// TIA Portal project "SkarabeuszURC" (V11)

(* hardware
DEVICE "SIMATIC 1200 station_1"  S71200.Device
   slot 0: "S7-1200 rack"  Rack  V1.0
   slot 1: "PLC_1"  CPU 1215C DC/DC/DC  6ES7 215-1AG31-0XB0  V3.0
   slot 2: "AI4 x 13 bits / AQ2 x 14 bits_1"  6ES7 234-4HE30-0XB0  V1.0
*)

// ===== PLC "PLC_1"  CPU 1215C DC/DC/DC =====

VAR_GLOBAL   // PLC tag table "Default tag table"
   "Tag_1" AT %QW0 : Word;
END_VAR

VAR_GLOBAL   // PLC tag table "Motor_Tags"
   "Motor_1_Pin_1" AT %Q0.0 : Bool;
   "Motor_1_Pin_2" AT %Q0.1 : Bool;
   "Motor_2_Pin_1" AT %Q0.2 : Bool;
   "Motor_2_Pin_2" AT %Q0.3 : Bool;
   "Motor_1_Analog" AT %QW96 : Int;
   "Motor_2_Analog" AT %QW98 : Int;
   "Motor_T_Pin_1" AT %Q0.4 : Bool;
   "Motor_T_Pin_2" AT %Q0.5 : Bool;
END_VAR

DATA_BLOCK "ModbusData"   // DB1
{ S7_Optimized_Access := 'FALSE' }
VERSION : 0.1
   VAR
      Registers : Array [1 .. 127] of Int;
      NDR : Bool;
      DR : Bool;
      ERROR : Bool;
      DISCONNECT : Bool;
      STATUS : Word;
   END_VAR
BEGIN
END_DATA_BLOCK

DATA_BLOCK "GlobalData"   // DB3
{ S7_Optimized_Access := 'FALSE' }
VERSION : 0.1
   VAR
      Motor_1_Direction : Word;
      Motor_2_Direction : Word;
      Motor_1_Speed : Word;
      Motor_2_Speed : Word;
      Motor_Turning_Direction : Word;
      Encoder_1_Data : Word;
      Encoder_2_Data : Word;
      Edge_1_Switch : Word;
      Edge_2_Switch : Word;
   END_VAR
   VAR RETAIN
      Forward_Direction : Word := 1;
   END_VAR
   VAR
      Backward_Direction : Word := 2;
      Break_Direction : Word := 3;
      Idle_Direction : Word := 4;
      Right_Turn : Word := 5;
      Left_Turn : Word := 6;
   END_VAR
BEGIN
END_DATA_BLOCK

// folder: System blocks/Program resources

DATA_BLOCK "IEC_Timer_0_DB_1"   // DB5
{ S7_Optimized_Access := 'FALSE' }
AUTHOR : Simatic
FAMILY : IEC
NAME : IEC_TMR
VERSION : 1.0
// stored: InstanceOfName ?
"?"
BEGIN
END_DATA_BLOCK

// folder: (top level)

FUNCTION "ModbusTCP" : Void   // FC1, LAD
{ S7_Optimized_Access := 'FALSE' }
VERSION : 0.1
BEGIN

REGION Network 1
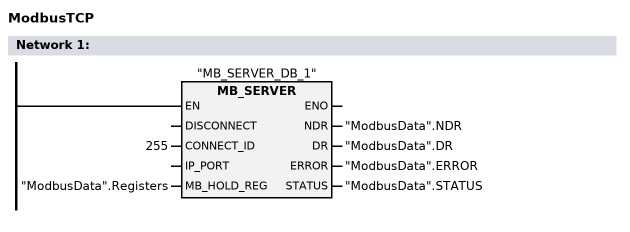
   "MB_SERVER_DB_1"(CONNECT_ID := 255,   // MB_SERVER
                    MB_HOLD_REG := "ModbusData".Registers,
                    NDR => "ModbusData".NDR,
                    DR => "ModbusData".DR,
                    ERROR => "ModbusData".ERROR,
                    STATUS => "ModbusData".STATUS);
END_REGION
END_FUNCTION

FUNCTION "Mapping" : Void   // FC2, LAD
{ S7_Optimized_Access := 'FALSE' }
VERSION : 0.1
BEGIN

REGION Network 1
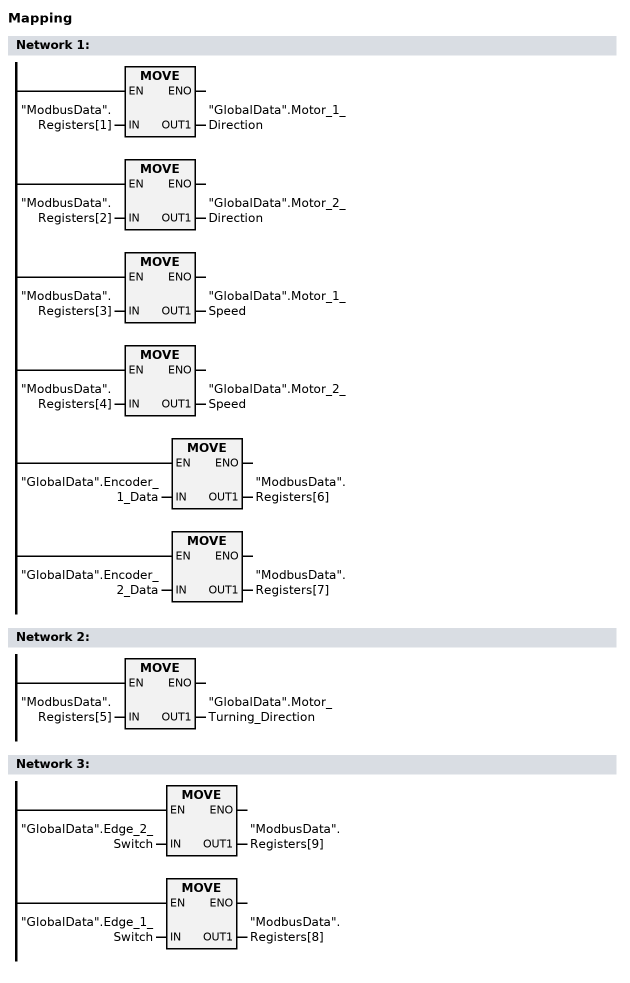
   RUNG wire#powerrail
      { S7_GenerateENO := "TRUE" } Move(in := "ModbusData".Registers[1], out1 => "GlobalData".Motor_1_Direction)
   END_RUNG
   RUNG wire#powerrail
      { S7_GenerateENO := "TRUE" } Move(in := "ModbusData".Registers[2], out1 => "GlobalData".Motor_2_Direction)
   END_RUNG
   RUNG wire#powerrail
      { S7_GenerateENO := "TRUE" } Move(in := "ModbusData".Registers[3], out1 => "GlobalData".Motor_1_Speed)
   END_RUNG
   RUNG wire#powerrail
      { S7_GenerateENO := "TRUE" } Move(in := "ModbusData".Registers[4], out1 => "GlobalData".Motor_2_Speed)
   END_RUNG
   RUNG wire#powerrail
      { S7_GenerateENO := "TRUE" } Move(in := "GlobalData".Encoder_1_Data, out1 => "ModbusData".Registers[6])
   END_RUNG
   RUNG wire#powerrail
      { S7_GenerateENO := "TRUE" } Move(in := "GlobalData".Encoder_2_Data, out1 => "ModbusData".Registers[7])
   END_RUNG
   // the same network as SCL:
   "GlobalData".Motor_1_Direction := "ModbusData".Registers[1];
   "GlobalData".Motor_2_Direction := "ModbusData".Registers[2];
   "GlobalData".Motor_1_Speed := "ModbusData".Registers[3];
   "GlobalData".Motor_2_Speed := "ModbusData".Registers[4];
   "ModbusData".Registers[6] := "GlobalData".Encoder_1_Data;
   "ModbusData".Registers[7] := "GlobalData".Encoder_2_Data;
END_REGION

REGION Network 2
   RUNG wire#powerrail
      { S7_GenerateENO := "TRUE" } Move(in := "ModbusData".Registers[5], out1 => "GlobalData".Motor_Turning_Direction)
   END_RUNG
   // the same network as SCL:
   "GlobalData".Motor_Turning_Direction := "ModbusData".Registers[5];
END_REGION

REGION Network 3
   RUNG wire#powerrail
      { S7_GenerateENO := "TRUE" } Move(in := "GlobalData".Edge_2_Switch, out1 => "ModbusData".Registers[9])
   END_RUNG
   RUNG wire#powerrail
      { S7_GenerateENO := "TRUE" } Move(in := "GlobalData".Edge_1_Switch, out1 => "ModbusData".Registers[8])
   END_RUNG
   // the same network as SCL:
   "ModbusData".Registers[9] := "GlobalData".Edge_2_Switch;
   "ModbusData".Registers[8] := "GlobalData".Edge_1_Switch;
END_REGION
END_FUNCTION

ORGANIZATION_BLOCK "Main"   // OB1, LAD, ProgramCycle
TITLE = "Main Program Sweep (Cycle)"
{ S7_Optimized_Access := 'FALSE' }
VERSION : 0.1
BEGIN
END_ORGANIZATION_BLOCK